// TIA Portal V17 export
// export: Created 2024-08-07T21:43:54.7016818Z, ExportSetting WithDefaults, DisplayName Totally Integrated Automation Portal, DisplayVersion V17 Update 7, DisplayName TIA Portal Openness, DisplayVersion V17 Update 7, DisplayName TIA Portal Version Control Interface, DisplayVersion V17, DisplayName SINAMICS Startdrive Advanced, DisplayVersion V17 SP2, DisplayName SINAMICS Startdrive G110M, G120, G120C, G120D, G120P, G115D, DisplayVersion V17 SP2, DisplayName SINAMICS Startdrive G130, G150, S120, S150, SINAMICS MV, S210, DisplayVersion V17 SP2, DisplayName STEP 7 Professional, DisplayVersion V17 Update 7, DisplayName STEP 7 Safety, DisplayVersion V17 Update 6, DisplayName WinCC Advanced / Unified PC, DisplayVersion V17 Update 7
FUNCTION_BLOCK "HydraulicCylinder"   // FB17, LAD
{ S7_Optimized_Access := 'TRUE' }
VERSION : 0.1
// stored: AutoNumber true, IsIECCheckEnabled false, IsRetainMemResEnabled false, MemoryReserve 100, SetENOAutomatically false, UDAEnableTagReadback false
   VAR_INPUT
      HydraulicActive : Bool;
      BasicPositionMin : Real;
      BasicPositionMax : Real;
      MaxPosition : Real;
      ManualCommand : Int;
      CylinderNumber : Int;
   END_VAR
   VAR_IN_OUT
      data : "UDT_HydraulicCylinderData";
   END_VAR
   VAR
      dataOld : "UDT_HydraulicCylinderData";
      noCollision { S7_SetPoint := 'True'} : Bool;
      IEC_Timer_0_Instance { S7_SetPoint := 'True'} : TON_TIME;
      R_TRIG_Instance { S7_SetPoint := 'True'} : R_TRIG;
      difference { S7_SetPoint := 'True'} : Real;
      re : Real;
      IEC_Timer_0_Instance_1 { S7_SetPoint := 'True'} : TON_TIME;
      RampFunction_Instance { S7_SetPoint := 'True'} : RampFunction;
      BasicPositionMin_1mm_margin : Real;
      BasicPositionMax_1mm_margin : Real;
   END_VAR
   VAR_TEMP
      command : Int;
   END_VAR
   VAR_TEMP   // added for the SCL form of the ladder/FBD networks
      _w1 : Bool;
   END_VAR
BEGIN

REGION Network 1
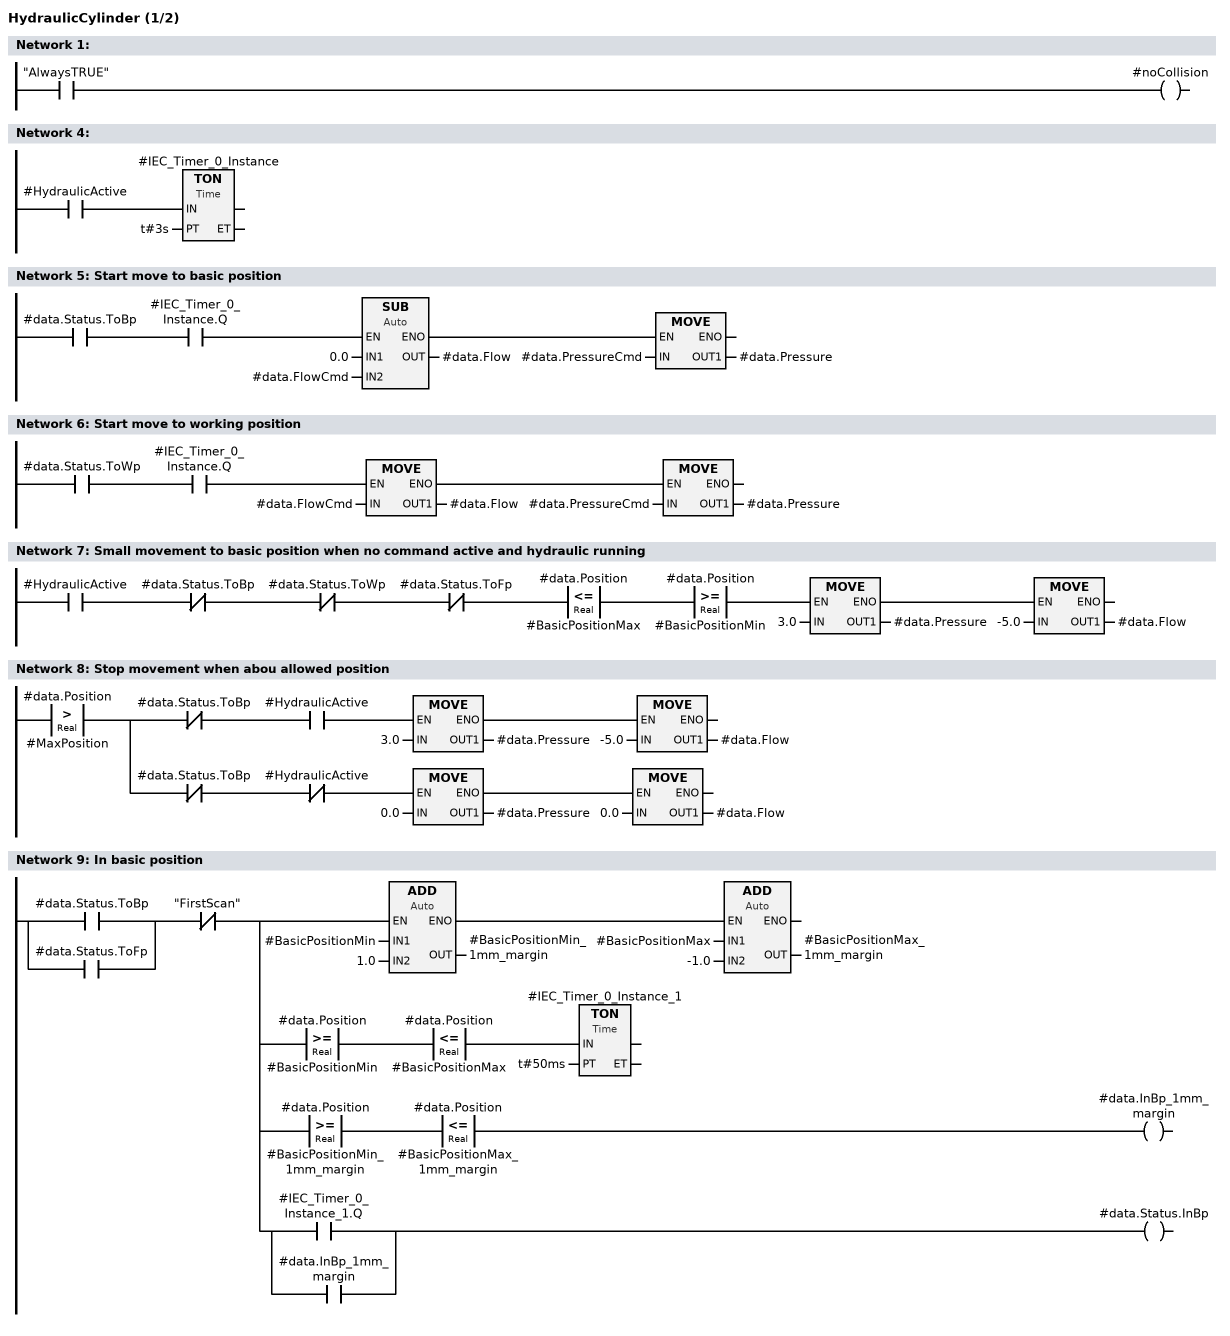
   RUNG wire#powerrail
      Contact( "AlwaysTRUE" )
      Coil( #noCollision )
   END_RUNG
   // the same network as SCL:
   #noCollision := "AlwaysTRUE";
END_REGION

REGION Network 2 (SCL)
   #command := #ManualCommand - #CylinderNumber;

   IF #command > 100 THEN
       "SandBoxData".MnualCommandMem := #command;
   END_IF;
   IF #command = 5000 THEN
       #data.Status.ToBp := true;
   END_IF;
   IF #command = 6000 THEN
       #data.Status.ToWp := true;
   END_IF;
   IF #command = 7000 THEN
       #data.Status.ToFp := true;
   END_IF;
END_REGION

REGION Network 3 (SCL): check new cylinder command
   //check if basic position req movement changed
   IF #data.Status.ToBp <> #dataOld.Status.ToBp AND #data.Status.ToBp THEN
       #data.Status.ToFp := false;
       #data.Status.ToWp := false;
       IF #noCollision THEN
           #data.Status.ToFp := false;
           #data.Status.ToWp := false;
       ELSE
           #data.Status.ToBp := false;
       END_IF;
   END_IF;
   //check if work position req movement changed
   IF #data.Status.ToWp <> #dataOld.Status.ToWp AND #data.Status.ToWp THEN
       IF #noCollision  THEN
           #data.Status.ToFp := false;
           #data.Status.ToBp := false;
       ELSE
           #data.Status.ToWp := false;
       END_IF;
   END_IF;
   //check if free position req movement changed
   IF #data.Status.ToFp <> #dataOld.Status.ToFp AND #data.Status.ToFp THEN
       #data.Status.ToBp := false;
       #data.Status.ToWp := false;
       IF #noCollision THEN
           #data.Status.ToBp := false;
           #data.Status.ToWp := false;
       ELSE
           #data.Status.ToFp := false;
       END_IF;
   END_IF;
   //store actual cylinder status to old
   #dataOld.Status := #data.Status;
END_REGION

REGION Network 4
   RUNG wire#powerrail
      Contact( #HydraulicActive )
      { S7_Templates := "time_type := Time" } #IEC_Timer_0_Instance.TON(pt := t#3s, et =>)
   END_RUNG
   // the same network as SCL:
   #IEC_Timer_0_Instance(IN := #HydraulicActive, PT := t#3s);   // TON
END_REGION

REGION Network 5: Start move to basic position
   RUNG wire#powerrail
      Contact( #data.Status.ToBp )
      Contact( #IEC_Timer_0_Instance.Q )
      Sub(in1 := 0.0, in2 := #data.FlowCmd, out => #data.Flow)
      Move(in := #data.PressureCmd, out1 => #data.Pressure)
   END_RUNG
   // the same network as SCL:
   IF #data.Status.ToBp AND #IEC_Timer_0_Instance.Q THEN
       #data.Flow := 0.0 - #data.FlowCmd;
       #data.Pressure := #data.PressureCmd;
   END_IF;
END_REGION

REGION Network 6: Start move to working position
   RUNG wire#powerrail
      Contact( #data.Status.ToWp )
      Contact( #IEC_Timer_0_Instance.Q )
      Move(in := #data.FlowCmd, out1 => #data.Flow)
      Move(in := #data.PressureCmd, out1 => #data.Pressure)
   END_RUNG
   // the same network as SCL:
   IF #data.Status.ToWp AND #IEC_Timer_0_Instance.Q THEN
       #data.Flow := #data.FlowCmd;
       #data.Pressure := #data.PressureCmd;
   END_IF;
END_REGION

REGION Network 7: Small movement to basic position when no command active and hydraulic running
   RUNG wire#powerrail
      Contact( #HydraulicActive )
      I_Contact( #data.Status.ToBp )
      I_Contact( #data.Status.ToWp )
      I_Contact( #data.Status.ToFp )
      { S7_Templates := "SrcType := Real" } LE_Contact(in1 := #data.Position, in2 := #BasicPositionMax)
      { S7_Templates := "SrcType := Real" } GE_Contact(in1 := #data.Position, in2 := #BasicPositionMin)
      Move(in := 3.0, out1 => #data.Pressure)
      Move(in := -5.0, out1 => #data.Flow)
   END_RUNG
   // the same network as SCL:
   IF #HydraulicActive AND NOT #data.Status.ToBp AND NOT #data.Status.ToWp AND NOT #data.Status.ToFp AND (#data.Position <= #BasicPositionMax) AND (#data.Position >= #BasicPositionMin) THEN
       #data.Pressure := 3.0;
       #data.Flow := -5.0;
   END_IF;
END_REGION

REGION Network 8: Stop movement when abou allowed position
   RUNG wire#powerrail
      { S7_Templates := "SrcType := Real" } GT_Contact(in1 := #data.Position, in2 := #MaxPosition)
      wire#w1
      I_Contact( #data.Status.ToBp )
      Contact( #HydraulicActive )
      Move(in := 3.0, out1 => #data.Pressure)
      Move(in := -5.0, out1 => #data.Flow)
   END_RUNG
   RUNG wire#w1
      I_Contact( #data.Status.ToBp )
      I_Contact( #HydraulicActive )
      Move(in := 0.0, out1 => #data.Pressure)
      Move(in := 0.0, out1 => #data.Flow)
   END_RUNG
   // the same network as SCL:
   #_w1 := #data.Position > #MaxPosition;
   IF #_w1 AND NOT #data.Status.ToBp AND #HydraulicActive THEN
       #data.Pressure := 3.0;
       #data.Flow := -5.0;
   END_IF;
   IF #_w1 AND NOT #data.Status.ToBp AND NOT #HydraulicActive THEN
       #data.Pressure := 0.0;
       #data.Flow := 0.0;
   END_IF;
END_REGION

REGION Network 9: In basic position
   RUNG wire#powerrail
      Contact( #data.Status.ToBp )
      wire#w1
      I_Contact( "FirstScan" )
      wire#w2
      Add(in1 := #BasicPositionMin, in2 := 1.0, out => #BasicPositionMin_1mm_margin)
      Add(in1 := #BasicPositionMax, in2 := -1.0, out => #BasicPositionMax_1mm_margin)
   END_RUNG
   RUNG wire#powerrail
      Contact( #data.Status.ToFp )
   END_RUNG wire#w1
   RUNG wire#w2
      { S7_Templates := "SrcType := Real" } GE_Contact(in1 := #data.Position, in2 := #BasicPositionMin)
      { S7_Templates := "SrcType := Real" } LE_Contact(in1 := #data.Position, in2 := #BasicPositionMax)
      { S7_Templates := "time_type := Time" } #IEC_Timer_0_Instance_1.TON(pt := t#50ms, et =>)
   END_RUNG
   RUNG wire#w2
      { S7_Templates := "SrcType := Real" } GE_Contact(in1 := #data.Position, in2 := #BasicPositionMin_1mm_margin)
      { S7_Templates := "SrcType := Real" } LE_Contact(in1 := #data.Position, in2 := #BasicPositionMax_1mm_margin)
      Coil( #data.InBp_1mm_margin )
   END_RUNG
   RUNG wire#w2
      Contact( #IEC_Timer_0_Instance_1.Q )
      wire#w3
      Coil( #data.Status.InBp )
   END_RUNG
   RUNG wire#w2
      Contact( #data.InBp_1mm_margin )
   END_RUNG wire#w3
   // the same network as SCL:
   #_w1 := (#data.Status.ToBp OR #data.Status.ToFp) AND NOT "FirstScan";
   IF #_w1 THEN
       #BasicPositionMin_1mm_margin := #BasicPositionMin + 1.0;
       #BasicPositionMax_1mm_margin := #BasicPositionMax + (-1.0);
   END_IF;
   #IEC_Timer_0_Instance_1(IN := #_w1 AND (#data.Position >= #BasicPositionMin) AND (#data.Position <= #BasicPositionMax),   // TON
                           PT := t#50ms);
   #data.InBp_1mm_margin := #_w1 AND (#data.Position >= #BasicPositionMin_1mm_margin) AND (#data.Position <= #BasicPositionMax_1mm_margin);
   #data.Status.InBp := #_w1 AND (#IEC_Timer_0_Instance_1.Q OR #data.InBp_1mm_margin);
END_REGION

REGION Network 10: Stand still - start stand still
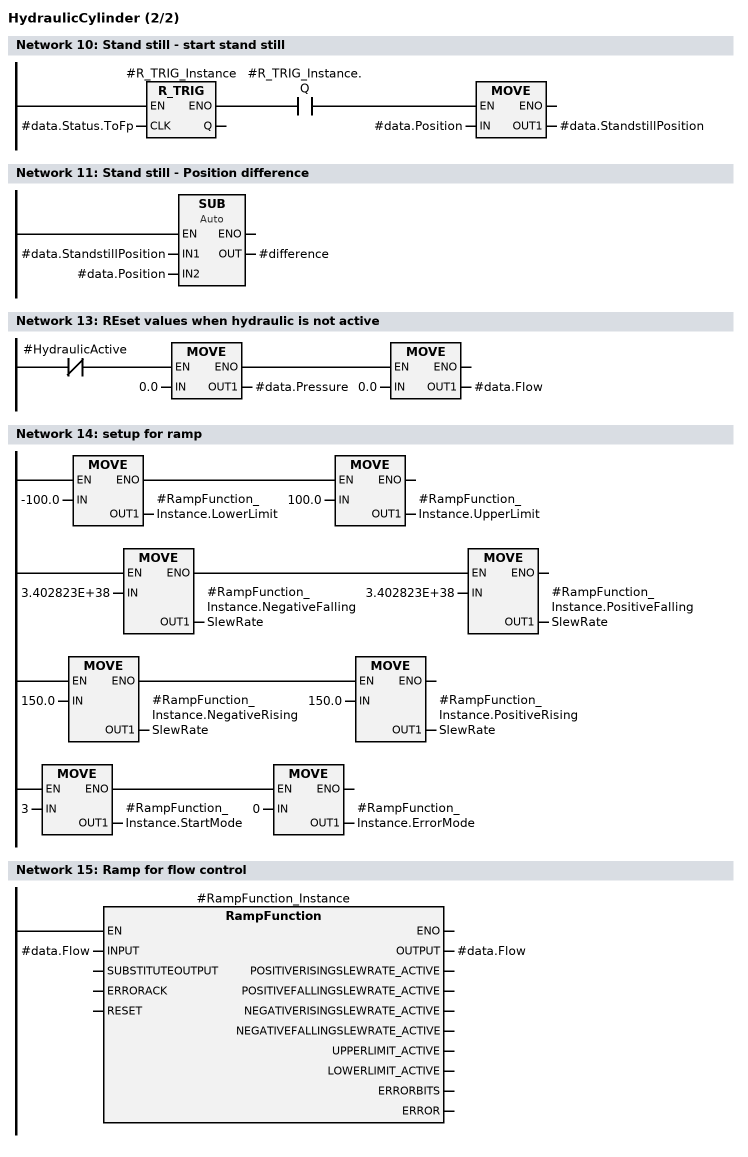
   RUNG wire#powerrail
      #R_TRIG_Instance.R_TRIG(CLK := #data.Status.ToFp, Q =>)
      Contact( #R_TRIG_Instance.Q )
      Move(in := #data.Position, out1 => #data.StandstillPosition)
   END_RUNG
   // the same network as SCL:
   #R_TRIG_Instance(CLK := #data.Status.ToFp, ENO => #_w1);   // R_TRIG
   IF #_w1 AND #R_TRIG_Instance.Q THEN #data.StandstillPosition := #data.Position; END_IF;
END_REGION

REGION Network 11: Stand still - Position difference
   RUNG wire#powerrail
      Sub(in1 := #data.StandstillPosition, in2 := #data.Position, out => #difference)
   END_RUNG
   // the same network as SCL:
   #difference := #data.StandstillPosition - #data.Position;
END_REGION

REGION Network 12 (SCL): Stand still - count regulation

   IF #data.Status.ToFp THEN
       #re := #difference;
       #re := #re * 10;
       IF #re > 0 THEN
           #re := #re + 5;
       END_IF;
       IF #re > 30 THEN
           #re := 30;
       END_IF;
       IF #re < -30 THEN
           #re := -30;
       END_IF;
       #data.Flow := #re;
       #data.Pressure := #data.PressureCmd;

       #data.Flow := 0;
       #data.Pressure := 0;

   END_IF;

   ;
END_REGION

REGION Network 13: REset values when hydraulic is not active
   RUNG wire#powerrail
      I_Contact( #HydraulicActive )
      Move(in := 0.0, out1 => #data.Pressure)
      Move(in := 0.0, out1 => #data.Flow)
   END_RUNG
   // the same network as SCL:
   IF NOT #HydraulicActive THEN
       #data.Pressure := 0.0;
       #data.Flow := 0.0;
   END_IF;
END_REGION

REGION Network 14: setup for ramp
   RUNG wire#powerrail
      Move(in := -100.0, out1 => #RampFunction_Instance.LowerLimit)
      Move(in := 100.0, out1 => #RampFunction_Instance.UpperLimit)
   END_RUNG
   RUNG wire#powerrail
      Move(in := 3.402823E+38, out1 => #RampFunction_Instance.NegativeFallingSlewRate)
      Move(in := 3.402823E+38, out1 => #RampFunction_Instance.PositiveFallingSlewRate)
   END_RUNG
   RUNG wire#powerrail
      Move(in := 150.0, out1 => #RampFunction_Instance.NegativeRisingSlewRate)
      Move(in := 150.0, out1 => #RampFunction_Instance.PositiveRisingSlewRate)
   END_RUNG
   RUNG wire#powerrail
      Move(in := 3, out1 => #RampFunction_Instance.StartMode)
      Move(in := 0, out1 => #RampFunction_Instance.ErrorMode)
   END_RUNG
   // the same network as SCL:
   #RampFunction_Instance.LowerLimit := -100.0;
   #RampFunction_Instance.UpperLimit := 100.0;
   #RampFunction_Instance.NegativeFallingSlewRate := 3.402823E+38;
   #RampFunction_Instance.PositiveFallingSlewRate := 3.402823E+38;
   #RampFunction_Instance.NegativeRisingSlewRate := 150.0;
   #RampFunction_Instance.PositiveRisingSlewRate := 150.0;
   #RampFunction_Instance.StartMode := 3;
   #RampFunction_Instance.ErrorMode := 0;
END_REGION

REGION Network 15: Ramp for flow control
   RUNG wire#powerrail
      #RampFunction_Instance.RampFunction(Input := #data.Flow, SubstituteOutput :=, ErrorAck :=, Reset :=, Output => #data.Flow, PositiveRisingSlewRate_Active =>, PositiveFallingSlewRate_Active =>, NegativeRisingSlewRate_Active =>, NegativeFallingSlewRate_Active =>, UpperLimit_Active =>, LowerLimit_Active =>, ErrorBits =>, Error =>)
   END_RUNG
   // the same network as SCL:
   #RampFunction_Instance(Input := #data.Flow, Output => #data.Flow);   // RampFunction
END_REGION
END_FUNCTION_BLOCK
